# EPICS substitutions: ek9000App/Db/EL1024_mbbiDirect.substitutions
file EL1024.template
{       pattern
        {
                TERMINAL,

        }
        {
        }
}
